% RSLogix 500 project PID_SUBTITUTE_LOGIC.RSS, saved by version 8.30.00.16 %
PROJECT "UNTITLED"    % processor: Bul.1763 MicroLogix 1100 Series B %

PROGRAM FILES
  LAD 2 "MAIN"  4 rungs
  LAD 3 "I/O"  3 rungs
  LAD 4 "CONTROL"  4 rungs
  LAD 5 "COMPUTE"  2 rungs

DATA FILES
  O0 OUTPUT  4 elements
  I1 INPUT  6 elements
  S2 STATUS  66 elements
  B3 BINARY  1 elements
  T4 TIMER  1 elements
  C5 COUNTER  1 elements
  R6 CONTROL  1 elements
  N7 INTEGER  7 elements
  F8 FLOAT  13 elements

LADDER 2 "MAIN"
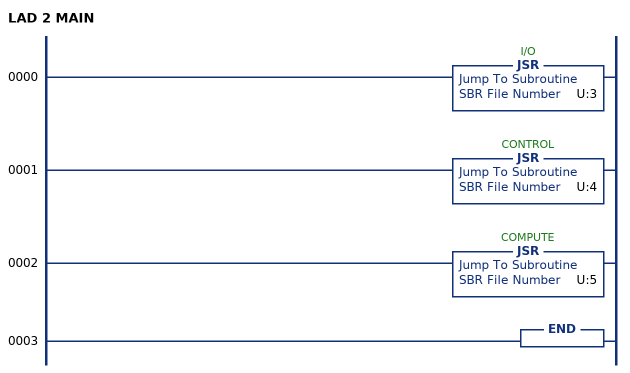
% Rung: 0 %
SOR JSR U:3 EOR
%   U:3  "I/O" %
% Rung: 1 %
SOR JSR U:4 EOR
%   U:4  "CONTROL" %
% Rung: 2 %
SOR JSR U:5 EOR
%   U:5  "COMPUTE" %
% Rung: 3 %
SOR END EOR

LADDER 3 "I/O"
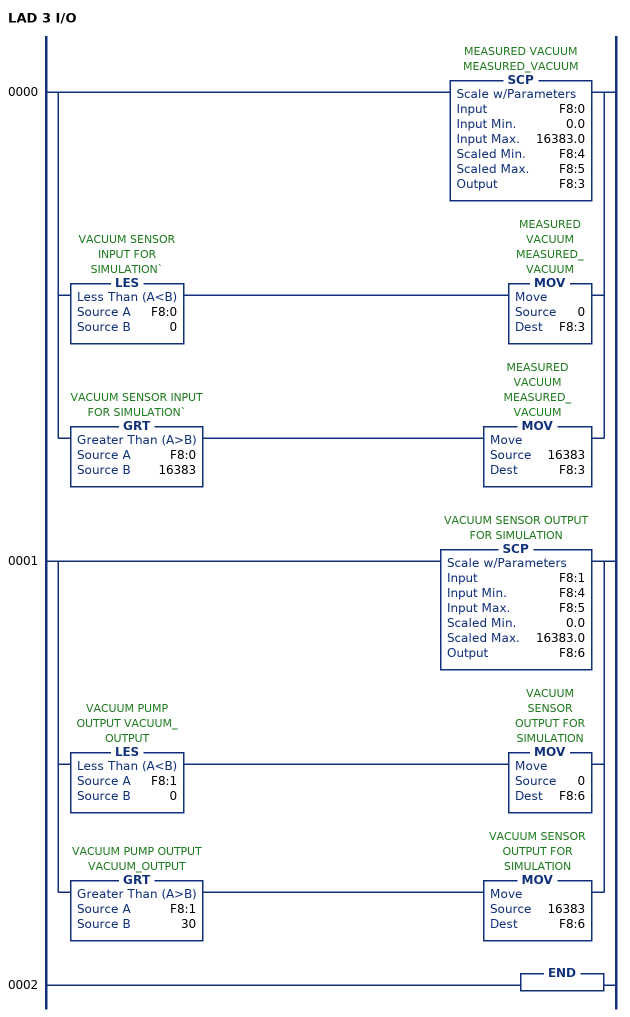
% Rung: 0 %
SOR BST SCP F8:0 0.0 16383.0 F8:4 F8:5 F8:3 NXB LES F8:0 0 MOV 0 F8:3 NXB GRT F8:0 16383 MOV 16383 F8:3 BND EOR
%   F8:0  "VACUUM SENSOR INPUT FOR SIMULATION`" %
%   F8:4  SENSOR_RANGE_MIN  "VACUUM SENSOR RANGE MINIMUM" %
%   F8:5  SENSOR_RANGE_MAX  "VACUUM SENSOR RANGE MAXIMUM" %
%   F8:3  MEASURED_VACUUM  "MEASURED VACUUM" %
% Rung: 1 %
SOR BST SCP F8:1 F8:4 F8:5 0.0 16383.0 F8:6 NXB LES F8:1 0 MOV 0 F8:6 NXB GRT F8:1 30 MOV 16383 F8:6 BND EOR
%   F8:1  VACUUM_OUTPUT  "VACUUM PUMP OUTPUT" %
%   F8:4  SENSOR_RANGE_MIN  "VACUUM SENSOR RANGE MINIMUM" %
%   F8:5  SENSOR_RANGE_MAX  "VACUUM SENSOR RANGE MAXIMUM" %
%   F8:6  "VACUUM SENSOR OUTPUT FOR SIMULATION" %
% Rung: 2 %
SOR END EOR

LADDER 4 "CONTROL"
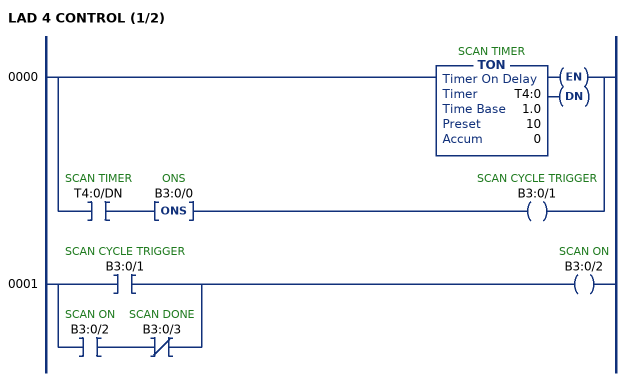
% Rung: 0 %
SOR BST TON T4:0 1.0 10 0 NXB XIC T4:0/DN ONS B3:0/0 OTE B3:0/1 BND EOR
%   T4:0  "SCAN TIMER" %
%   T4:0/DN  "SCAN TIMER" %
%   B3:0/0  "ONS" %
%   B3:0/1  "SCAN CYCLE TRIGGER" %
% Rung: 1 %
SOR BST XIC B3:0/1 NXB XIC B3:0/2 XIO B3:0/3 BND OTE B3:0/2 EOR
%   B3:0/1  "SCAN CYCLE TRIGGER" %
%   B3:0/2  "SCAN ON" %
%   B3:0/3  "SCAN DONE" %

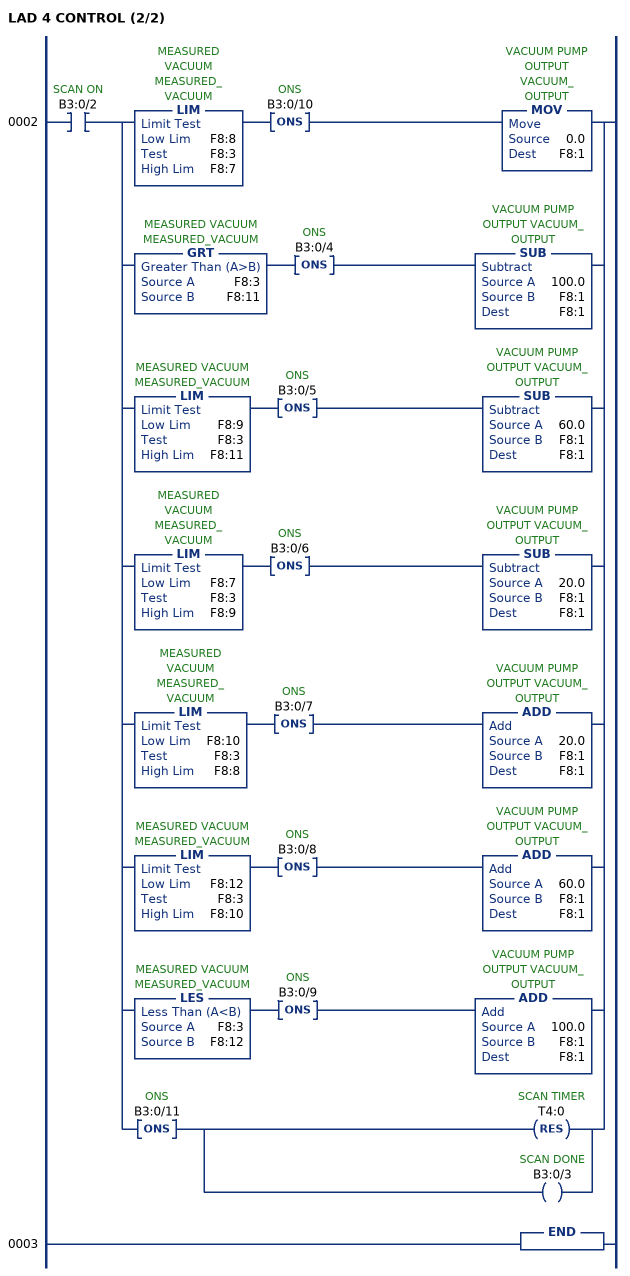
% Rung: 2 %
SOR XIC B3:0/2 BST LIM F8:8 F8:3 F8:7 ONS B3:0/10 MOV 0.0 F8:1 NXB GRT F8:3 F8:11 ONS B3:0/4 SUB 100.0 F8:1 F8:1 NXB LIM F8:9 F8:3 F8:11 ONS B3:0/5 SUB 60.0 F8:1 F8:1 NXB LIM F8:7 F8:3 F8:9 ONS B3:0/6 SUB 20.0 F8:1 F8:1 NXB LIM F8:10 F8:3 F8:8 ONS B3:0/7 ADD 20.0 F8:1 F8:1 NXB LIM F8:12 F8:3 F8:10 ONS B3:0/8 ADD 60.0 F8:1 F8:1 NXB LES F8:3 F8:12 ONS B3:0/9 ADD 100.0 F8:1 F8:1 NXB ONS B3:0/11 BST RES T4:0 NXB OTE B3:0/3 BND BND EOR
%   B3:0/2  "SCAN ON" %
%   F8:8  "COMPARE VALUE -4%" %
%   F8:3  MEASURED_VACUUM  "MEASURED VACUUM" %
%   F8:7  "COMPARE VALUE +4%" %
%   B3:0/10  "ONS" %
%   F8:1  VACUUM_OUTPUT  "VACUUM PUMP OUTPUT" %
%   F8:11  "COMPARE VALUE +30%" %
%   B3:0/4  "ONS" %
%   F8:9  "COMPARE VALUE +15%" %
%   B3:0/5  "ONS" %
%   B3:0/6  "ONS" %
%   F8:10  "COMPARE VALUE -15%" %
%   B3:0/7  "ONS" %
%   F8:12  "COMPARE VALUE -30%" %
%   B3:0/8  "ONS" %
%   B3:0/9  "ONS" %
%   B3:0/11  "ONS" %
%   T4:0  "SCAN TIMER" %
%   B3:0/3  "SCAN DONE" %
% Rung: 3 %
SOR END EOR

LADDER 5 "COMPUTE"
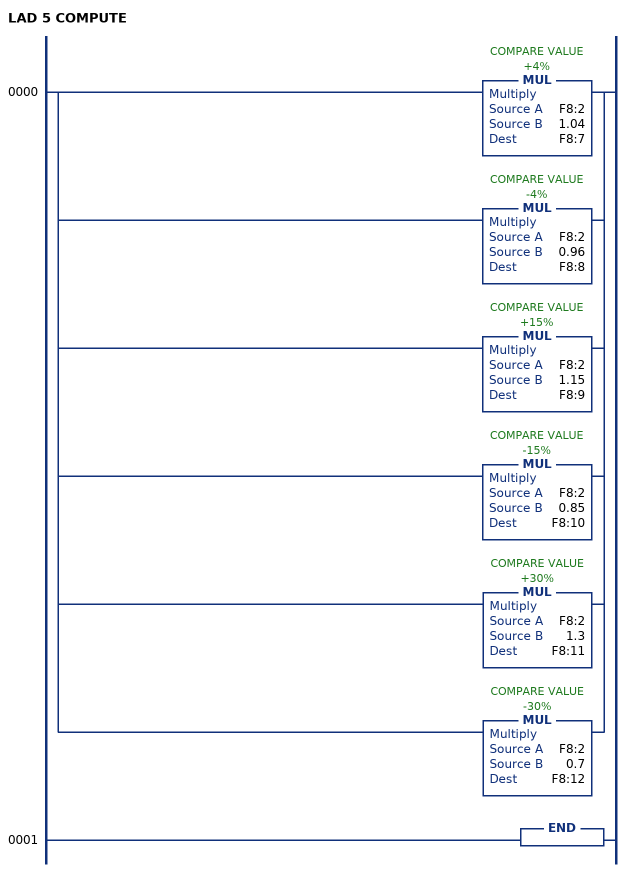
% Rung: 0 %
SOR BST MUL F8:2 1.04 F8:7 NXB MUL F8:2 0.96 F8:8 NXB MUL F8:2 1.15 F8:9 NXB MUL F8:2 0.85 F8:10 NXB MUL F8:2 1.3 F8:11 NXB MUL F8:2 0.7 F8:12 BND EOR
%   F8:2  VACUUM_SETPOINT  "VACUUM SETPOINT" %
%   F8:7  "COMPARE VALUE +4%" %
%   F8:8  "COMPARE VALUE -4%" %
%   F8:9  "COMPARE VALUE +15%" %
%   F8:10  "COMPARE VALUE -15%" %
%   F8:11  "COMPARE VALUE +30%" %
%   F8:12  "COMPARE VALUE -30%" %
% Rung: 1 %
SOR END EOR

OTHER DOCUMENTED ADDRESSES
  MOV  

DATA TABLE (non-zero values as saved)
DATA T4
% .PRE .ACC %
% T4:0 % 10 0
DATA F8
% F8:0 % 0 0 15 0 0
% F8:5 % 30 0 0 0 0
